// TIA Portal V17 export
// export: Created 2025-03-05T08:02:10.5039967Z, ExportSetting WithDefaults, DisplayName Totally Integrated Automation Portal, DisplayVersion V17 Update 8, DisplayName TIA Portal Openness, DisplayVersion V17 Update 8, DisplayName TIA Portal Version Control Interface, DisplayVersion V17, DisplayName SINAMICS Startdrive Advanced, DisplayVersion V17 SP2, DisplayName SINAMICS Startdrive G110M, G120, G120C, G120D, G120P, G115D, DisplayVersion V17 SP2, DisplayName SINAMICS Startdrive G130, G150, S120, S150, SINAMICS MV, S210, DisplayVersion V17 SP2, DisplayName STEP 7 Professional, DisplayVersion V17 Update 8, DisplayName SINUMERIK ONE STEP 7 Toolbox, DisplayVersion V17 Update 12, DisplayName SINUMERIK 840D sl STEP 7 Toolbox, DisplayVersion V17 Update 12, DisplayName STEP 7 Safety, DisplayVersion V17 Update 6, DisplayName WinCC Advanced, DisplayVersion V17 Update 8
TYPE "READ_AXES_POSITIONS_CH"
// stored: IsFailsafeCompliant false
   STRUCT
      READING_FAULT_1 : Bool;   // READING FAULT 1
      READING_DONE_1 : Bool;   // READING DONE 1
      REQUEST_1 : Bool;   // REQUEST 1
      READING_FAULT_2 : Bool;   // READING FAULT 2
      READING_DONE_2 : Bool;   // READING DONE 2
      REQUEST_2 : Bool;   // REQUEST 2
      READING_FAULT_3 : Bool;   // READING FAULT 3
      READING_DONE_3 : Bool;   // READING DONE 3
      REQUEST_3 : Bool;   // REQUEST 3
      FAULT_1 : Bool;   // FAULT 1
      FAULT_2 : Bool;   // FAULT 2
      FAULT_3 : Bool;   // FAULT 3
      IS : Bool;   // INMEDIATE STOP ALARMS / IMMEDIATE STOP ALARMS
      IS_SEOC : Bool;   // INMEDIATE STOP & STOP END OF CYCLE ALARMS / IMMEDIATE STOP & STOP END OF CYCLE ALARMS
      RHP : Bool;   // RETURN HOME POSITION ALARMS
      RHP_SEOC : Bool;   // RETURN HOME POSITION & STOP END OF CYCLE ALARMS
      SEOC : Bool;   // STOP END OF CYCLE ALARMS
      IS_WARNING : Bool;   // INMEDIATE STOP WARNING / IMMEDIATE STOP WARNING
      RHP_WARNING : Bool;   // RETURN HOME POSITION WARNING
      SEOC_WARNING : Bool;   // STOP END OF CYCLE WARNING
      WARNINGS : Bool;   // WARNINGS
      Help : Bool;   // Help
      Aux : Bool;   // Aux
      Aux1 : Bool;   // Aux1
      Aux2 : Bool;   // Aux2
      Aux3 : Bool;   // Aux3
      Aux4 : Bool;   // Aux4
      Aux5 : Bool;   // Aux5
      Aux6 : Bool;   // Aux6
      Aux7 : Bool;   // Aux7
      READING_STATUS : Word;   // READING STATUS
      POSITION_AXIS_1 : DWord;   // POSITION AXIS 1
      POSITION_AXIS_2 : DWord;   // POSITION AXIS 2
      POSITION_AXIS_3 : DWord;   // POSITION AXIS 3
      POSITION_AXIS_4 : DWord;   // POSITION AXIS 4
      POSITION_AXIS_5 : DWord;   // POSITION AXIS 5
      POSITION_AXIS_6 : DWord;   // POSITION AXIS 6
      POSITION_AXIS_7 : DWord;   // POSITION AXIS 7
      POSITION_AXIS_8 : DWord;   // POSITION AXIS 8
      POSITION_AXIS_9 : DWord;   // POSITION AXIS 9
      POSITION_AXIS_10 : DWord;   // POSITION AXIS 10
      POSITION_AXIS_11 : DWord;   // POSITION AXIS 11
      POSITION_AXIS_12 : DWord;   // POSITION AXIS 12
      POSITION_AXIS_13 : DWord;   // POSITION AXIS 13
      POSITION_AXIS_14 : DWord;   // POSITION AXIS 14
      POSITION_AXIS_15 : DWord;   // POSITION AXIS 15
      POSITION_AXIS_16 : DWord;   // POSITION AXIS 16
      POSITION_AXIS_17 : DWord;   // POSITION AXIS 17
      POSITION_AXIS_18 : DWord;   // POSITION AXIS 18
      POSITION_AXIS_19 : DWord;   // POSITION AXIS 19
      POSITION_AXIS_20 : DWord;   // POSITION AXIS 20
      CH_Reading_1 : Struct   // CH Reading 1
         SYNTAX_ID : Byte := BYTE#16#82;   // SYNTAX ID
         Area_Unit : Byte := BYTE#16#41;   // Area_Unit
         Column : Word := WORD#16#0002;   // Column
         Line : Word := WORD#16#0001;   // Line
         BlockType : Byte := BYTE#16#74;   // Block Type
         NumOfLine : Byte := BYTE#16#01;   // Number Of Line
         DataType : Byte := BYTE#16#0F;   // Data Type
         Length : Byte := BYTE#16#08;   // Length
      END_STRUCT;
      CH_Reading_2 : Struct   // CH Reading 2
         SYNTAX_ID : Byte := BYTE#16#82;   // SYNTAX ID
         Area_Unit : Byte := BYTE#16#41;   // Area_Unit
         Column : Word := WORD#16#0002;   // Column
         Line : Word := WORD#16#0002;   // Line
         BlockType : Byte := BYTE#16#74;   // Block Type
         NumOfLine : Byte := BYTE#16#01;   // Number Of Line
         DataType : Byte := BYTE#16#0F;   // Data Type
         Length : Byte := BYTE#16#08;   // Length
      END_STRUCT;
      CH_Reading_3 : Struct   // CH Reading 3
         SYNTAX_ID : Byte := BYTE#16#82;   // SYNTAX ID
         Area_Unit : Byte := BYTE#16#41;   // Area_Unit
         Column : Word := WORD#16#0002;   // Column
         Line : Word := WORD#16#0003;   // Line
         BlockType : Byte := BYTE#16#74;   // Block Type
         NumOfLine : Byte := BYTE#16#01;   // Number Of Line
         DataType : Byte := BYTE#16#0F;   // Data Type
         Length : Byte := BYTE#16#08;   // Length
      END_STRUCT;
      CH_Reading_4 : Struct   // CH Reading 4
         SYNTAX_ID : Byte := BYTE#16#82;   // SYNTAX ID
         Area_Unit : Byte := BYTE#16#41;   // Area_Unit
         Column : Word := WORD#16#0002;   // Column
         Line : Word := WORD#16#0004;   // Line
         BlockType : Byte := BYTE#16#74;   // Block Type
         NumOfLine : Byte := BYTE#16#01;   // Number Of Line
         DataType : Byte := BYTE#16#0F;   // Data Type
         Length : Byte := BYTE#16#08;   // Length
      END_STRUCT;
      CH_Reading_5 : Struct   // CH Reading 5
         SYNTAX_ID : Byte := BYTE#16#82;   // SYNTAX ID
         Area_Unit : Byte := BYTE#16#41;   // Area_Unit
         Column : Word := WORD#16#0002;   // Column
         Line : Word := WORD#16#0005;   // Line
         BlockType : Byte := BYTE#16#74;   // Block Type
         NumOfLine : Byte := BYTE#16#01;   // Number Of Line
         DataType : Byte := BYTE#16#0F;   // Data Type
         Length : Byte := BYTE#16#08;   // Length
      END_STRUCT;
      CH_Reading_6 : Struct   // CH Reading 6
         SYNTAX_ID : Byte := BYTE#16#82;   // SYNTAX ID
         Area_Unit : Byte := BYTE#16#41;   // Area_Unit
         Column : Word := WORD#16#0002;   // Column
         Line : Word := WORD#16#0006;   // Line
         BlockType : Byte := BYTE#16#74;   // Block Type
         NumOfLine : Byte := BYTE#16#01;   // Number Of Line
         DataType : Byte := BYTE#16#0F;   // Data Type
         Length : Byte := BYTE#16#08;   // Length
      END_STRUCT;
      CH_Reading_7 : Struct   // CH Reading 7
         SYNTAX_ID : Byte := BYTE#16#82;   // SYNTAX ID
         Area_Unit : Byte := BYTE#16#41;   // Area_Unit
         Column : Word := WORD#16#0002;   // Column
         Line : Word := WORD#16#0007;   // Line
         BlockType : Byte := BYTE#16#74;   // Block Type
         NumOfLine : Byte := BYTE#16#01;   // Number Of Line
         DataType : Byte := BYTE#16#0F;   // Data Type
         Length : Byte := BYTE#16#08;   // Length
      END_STRUCT;
      CH_Reading_8 : Struct   // CH Reading 8
         SYNTAX_ID : Byte := BYTE#16#82;   // SYNTAX ID
         Area_Unit : Byte := BYTE#16#41;   // Area_Unit
         Column : Word := WORD#16#0002;   // Column
         Line : Word := WORD#16#0008;   // Line
         BlockType : Byte := BYTE#16#74;   // Block Type
         NumOfLine : Byte := BYTE#16#01;   // Number Of Line
         DataType : Byte := BYTE#16#0F;   // Data Type
         Length : Byte := BYTE#16#08;   // Length
      END_STRUCT;
      CH_Reading_9 : Struct   // CH Reading 9
         SYNTAX_ID : Byte := BYTE#16#82;   // SYNTAX ID
         Area_Unit : Byte := BYTE#16#41;   // Area_Unit
         Column : Word := WORD#16#0002;   // Column
         Line : Word := WORD#16#0009;   // Line
         BlockType : Byte := BYTE#16#74;   // Block Type
         NumOfLine : Byte := BYTE#16#01;   // Number Of Line
         DataType : Byte := BYTE#16#0F;   // Data Type
         Length : Byte := BYTE#16#08;   // Length
      END_STRUCT;
      CH_Reading_10 : Struct   // CH Reading 10
         SYNTAX_ID : Byte := BYTE#16#82;   // SYNTAX ID
         Area_Unit : Byte := BYTE#16#41;   // Area_Unit
         Column : Word := WORD#16#0002;   // Column
         Line : Word := WORD#16#000A;   // Line
         BlockType : Byte := BYTE#16#73;   // Block Type
         NumOfLine : Byte := BYTE#16#01;   // Number Of Line
         DataType : Byte := BYTE#16#0F;   // Data Type
         Length : Byte := BYTE#16#08;   // Length
      END_STRUCT;
      CH_Reading_11 : Struct   // CH Reading 11
         SYNTAX_ID : Byte := BYTE#16#82;   // SYNTAX ID
         Area_Unit : Byte := BYTE#16#41;   // Area_Unit
         Column : Word := WORD#16#0002;   // Column
         Line : Word := WORD#16#000B;   // Line
         BlockType : Byte := BYTE#16#74;   // Block Type
         NumOfLine : Byte := BYTE#16#01;   // Number Of Line
         DataType : Byte := BYTE#16#0F;   // Data Type
         Length : Byte := BYTE#16#08;   // Length
      END_STRUCT;
      CH_Reading_12 : Struct   // CH Reading 12
         SYNTAX_ID : Byte := BYTE#16#82;   // SYNTAX ID
         Area_Unit : Byte := BYTE#16#41;   // Area_Unit
         Column : Word := WORD#16#0002;   // Column
         Line : Word := WORD#16#000C;   // Line
         BlockType : Byte := BYTE#16#74;   // Block Type
         NumOfLine : Byte := BYTE#16#01;   // Number Of Line
         DataType : Byte := BYTE#16#0F;   // Data Type
         Length : Byte := BYTE#16#08;   // Length
      END_STRUCT;
      CH_Reading_13 : Struct   // CH Reading 13
         SYNTAX_ID : Byte := BYTE#16#82;   // SYNTAX ID
         Area_Unit : Byte := BYTE#16#41;   // Area_Unit
         Column : Word := WORD#16#0002;   // Column
         Line : Word := WORD#16#000D;   // Line
         BlockType : Byte := BYTE#16#74;   // Block Type
         NumOfLine : Byte := BYTE#16#01;   // Number Of Line
         DataType : Byte := BYTE#16#0F;   // Data Type
         Length : Byte := BYTE#16#08;   // Length
      END_STRUCT;
      CH_Reading_14 : Struct   // CH Reading 14
         SYNTAX_ID : Byte := BYTE#16#82;   // SYNTAX ID
         Area_Unit : Byte := BYTE#16#41;   // Area_Unit
         Column : Word := WORD#16#0002;   // Column
         Line : Word := WORD#16#000E;   // Line
         BlockType : Byte := BYTE#16#74;   // Block Type
         NumOfLine : Byte := BYTE#16#01;   // Number Of Line
         DataType : Byte := BYTE#16#0F;   // Data Type
         Length : Byte := BYTE#16#08;   // Length
      END_STRUCT;
      CH_Reading_15 : Struct   // CH Reading 15
         SYNTAX_ID : Byte := BYTE#16#82;   // SYNTAX ID
         Area_Unit : Byte := BYTE#16#41;   // Area_Unit
         Column : Word := WORD#16#0002;   // Column
         Line : Word := WORD#16#000F;   // Line
         BlockType : Byte := BYTE#16#74;   // Block Type
         NumOfLine : Byte := BYTE#16#01;   // Number Of Line
         DataType : Byte := BYTE#16#0F;   // Data Type
         Length : Byte := BYTE#16#08;   // Length
      END_STRUCT;
      CH_Reading_16 : Struct   // CH Reading 16
         SYNTAX_ID : Byte := BYTE#16#82;   // SYNTAX ID
         Area_Unit : Byte := BYTE#16#41;   // Area_Unit
         Column : Word := WORD#16#0002;   // Column
         Line : Word := WORD#16#0010;   // Line
         BlockType : Byte := BYTE#16#74;   // Block Type
         NumOfLine : Byte := BYTE#16#01;   // Number Of Line
         DataType : Byte := BYTE#16#0F;   // Data Type
         Length : Byte := BYTE#16#08;   // Length
      END_STRUCT;
      CH_Reading_17 : Struct   // CH Reading 17
         SYNTAX_ID : Byte := BYTE#16#82;   // SYNTAX ID
         Area_Unit : Byte := BYTE#16#41;   // Area_Unit
         Column : Word := WORD#16#0002;   // Column
         Line : Word := WORD#16#0011;   // Line
         BlockType : Byte := BYTE#16#74;   // Block Type
         NumOfLine : Byte := BYTE#16#01;   // Number Of Line
         DataType : Byte := BYTE#16#0F;   // Data Type
         Length : Byte := BYTE#16#08;   // Length
      END_STRUCT;
      CH_Reading_18 : Struct   // CH Reading 18
         SYNTAX_ID : Byte := BYTE#16#82;   // SYNTAX ID
         Area_Unit : Byte := BYTE#16#41;   // Area_Unit
         Column : Word := WORD#16#0002;   // Column
         Line : Word := WORD#16#0012;   // Line
         BlockType : Byte := BYTE#16#74;   // Block Type
         NumOfLine : Byte := BYTE#16#01;   // Number Of Line
         DataType : Byte := BYTE#16#0F;   // Data Type
         Length : Byte := BYTE#16#08;   // Length
      END_STRUCT;
      CH_Reading_19 : Struct   // CH Reading 19
         SYNTAX_ID : Byte := BYTE#16#82;   // SYNTAX ID
         Area_Unit : Byte := BYTE#16#41;   // Area_Unit
         Column : Word := WORD#16#0002;   // Column
         Line : Word := WORD#16#0013;   // Line
         BlockType : Byte := BYTE#16#74;   // Block Type
         NumOfLine : Byte := BYTE#16#01;   // Number Of Line
         DataType : Byte := BYTE#16#0F;   // Data Type
         Length : Byte := BYTE#16#08;   // Length
      END_STRUCT;
      CH_Reading_20 : Struct   // CH Reading 20
         SYNTAX_ID : Byte := BYTE#16#82;   // SYNTAX ID
         Area_Unit : Byte := BYTE#16#41;   // Area_Unit
         Column : Word := WORD#16#0002;   // Column
         Line : Word := WORD#16#0014;   // Line
         BlockType : Byte := BYTE#16#74;   // Block Type
         NumOfLine : Byte := BYTE#16#01;   // Number Of Line
         DataType : Byte := BYTE#16#0F;   // Data Type
         Length : Byte := BYTE#16#08;   // Length
      END_STRUCT;
   END_STRUCT;
END_TYPE
